KUKA KRL program: chk_w9_wechs_ok.src

&ACCESS RV5
&COMMENT Gripper Axor 903
DEF chk_w9_wechs_ok( )

; VERIFICAÇÃO DE FERRAMENTA: GRIPPER Axor 903

$TIMER[10] = 0
$TIMER_STOP[10] = FALSE

wait for ((NOT $IN[577]) and ($IN[585]) and ($in[161]) and ($in[177]) and ($in[193]) and ($in[201]) and ($in[209]) and ($IN[169]) and ($in[185]) AND ($in[219]))

$TIMER_STOP[10] = TRUE
$TIMER[10] = 0

;//---- End -------
;Diag_Appl(#Off,5)

END
